FUNCTION_BLOCK FB_Transport
VAR_INPUT
	bEnable : BOOL;
	bExecute : BOOL;
	nstation : INT;
	//Hardware Eingänge
	bSens1 : BOOL;
	bSens2 : BOOL;
	bSens3 : BOOL;
	bSens4 : BOOL;
END_VAR
VAR_OUTPUT
	eState : eBetriebszustand;
	bstopper1 : BOOL;
	bstopper2 : BOOL;
	bstopper3 : BOOL;
	
END_VAR
VAR
	fbTransportE : FB_TransportE;
	fbTransportLogik : FB_TransportLogik;
	fbTransportBand : FB_Foerderband;
	fbTransportA : FB_TransportA;
END_VAR
VAR_IN_OUT
	//Achsenreferenz
	ax : Axis_Ref;
END_VAR

fbTransportE(
	bSens1:= bSens1, 
	bSens2:= bSens2, 
	bSens3:= bSens3, 
	bSens4:= bSens4, 
	bStation1=> , 
	bStation2=> , 
	bStation3=> , 
	bStation4=> );
	
fbTransportLogik(
	bEnable:= bEnable, 
	bExecute:= bExecute, 
	eStateE:= fbTransportBand.estate, 
	nStation:= nstation, 
	bStation1:= fbTransportE.bStation1, 
	bStation2:= fbTransportE.bStation2, 
	bStation3:= fbTransportE.bStation3, 
	bStation4:= fbTransportE.bStation4, 
	bEnableA=> , 
	bExecuteA=> ,  
	bStop1=> , 
	bStop2=> , 
	bStop3=> , 
	bStop4=> );
	
fbTransportBand(
	benable:= fbTransportLogik.bEnableA, 
	bexecute:= fbTransportLogik.bExecuteA, 
	bhalt:= fbTransportLogik.bStopA, 
	estate=> , 
	ax:= ax);
	
fbTransportA(
	bstop1:= fbTransportLogik.bStop1, 
	bstop2:= fbTransportLogik.bStop2, 
	bstop3:= fbTransportLogik.bStop3, 
	bstopper1=> bStopper1, 
	bstopper2=> bStopper2, 
	bstopper3=> bStopper3);

END_FUNCTION_BLOCK

(* stored: Version 1.1.0.1, ProductVersion 3.1.4024.15
   POU FB_Transport: Id {2b71af40-e306-4ae2-a807-c5fa554971f8}, SpecialFunc None *)
